TYPE HandlingComSubscribe :
STRUCT
  Request : HandlingComRequest; // contains booleans that are used to start a specific sequence.
  Equipment : HandlingComSubscribeEquipment;  // structs for equipment objects which are used by the bridges
END_STRUCT
END_TYPE

(* stored: Version 1.1.0.1
   DUT HandlingComSubscribe: Id {2e32f878-89e1-46ab-98f4-01c1f6554eea} *)
